FUNCTION_BLOCK FB_DCControl
VAR_INPUT
END_VAR
VAR_OUTPUT
END_VAR
VAR
END_VAR

END_FUNCTION_BLOCK

(* stored: Version 1.1.0.1, ProductVersion 3.1.4024.10
   POU FB_DCControl: Id {8c229838-3742-48b4-a907-91e08ed4966e}, SpecialFunc None *)
